// TIA Portal V15.1 export
// export: Created 2024-06-21T08:40:53.4575438Z, ExportSetting WithDefaults, DisplayName Totally Integrated Automation Portal, DisplayVersion V15.1 Update 5, DisplayName TIA Portal Openness, DisplayVersion V15.1 Update 5, DisplayName SINAMICS Startdrive Advanced, DisplayVersion V15.1, DisplayName G130, G150, S120, S150, SINAMICS MV, S210, DisplayVersion V15.1, DisplayName G110M, G120, G120C, G120D, G120P, DisplayVersion V15.1, DisplayName STEP 7 Professional, DisplayVersion V15.1 Update 5, DisplayName STEP 7 Safety, DisplayVersion V15.1, DisplayName WinCC Professional, DisplayVersion V15.1 Update 5, DisplayName SIMATIC Visualization Architect, DisplayVersion V15.1
FUNCTION_BLOCK "LConditionDelay"   // FB1101, FBD
TITLE = LConditionDelay
{ S7_Optimized_Access := 'FALSE' }
VERSION : 0.1
// stored: AutoNumber false, IsIECCheckEnabled false, SetENOAutomatically False, UDAEnableTagReadback false
   VAR_INPUT
      I_Condition { ExternalAccessible := 'False'; ExternalVisible := 'False'; ExternalWritable := 'False'} : Bool;   // Condition
      I_ExtDelayTime { ExternalAccessible := 'False'; ExternalVisible := 'False'; ExternalWritable := 'False'} : DInt;   // External delay time
      I_ActivedExtDelayTime { ExternalAccessible := 'False'; ExternalVisible := 'False'; ExternalWritable := 'False'} : Bool;   // Activated external delay time
      I_HoldCond { ExternalAccessible := 'False'; ExternalVisible := 'False'; ExternalWritable := 'False'} : Bool;   // Hold condition normal open
      I_ResetCond { ExternalAccessible := 'False'; ExternalVisible := 'False'; ExternalWritable := 'False'} : Bool;   // Reset condition normal open
      I_BypassCond { ExternalAccessible := 'False'; ExternalVisible := 'False'; ExternalWritable := 'False'} : Bool;   // Bypass condition normal open
   END_VAR
   VAR_OUTPUT
      O_ConditionDelayed { ExternalAccessible := 'False'; ExternalVisible := 'False'; ExternalWritable := 'False'} : Bool;   // Condition delayed
   END_VAR
   VAR_IN_OUT
      H_HMI : "H_HMI";   // Animation
      H_ConditionDelay : "H_ConditionDelay";   // Animation
   END_VAR
   VAR DB_SPECIFIC
      TimerResult { ExternalAccessible := 'False'; ExternalVisible := 'False'; ExternalWritable := 'False'} : Bool;   // Timer result
      TimerValue { ExternalAccessible := 'False'; ExternalVisible := 'False'; ExternalWritable := 'False'} : DInt;   // Timer value
      TimerValueElapsed { ExternalAccessible := 'False'; ExternalVisible := 'False'; ExternalWritable := 'False'} : DInt;   // Timer value elapsed
      TimerExtValue { ExternalAccessible := 'False'; ExternalVisible := 'False'; ExternalWritable := 'False'} : DInt;   // Timer external value
      PrevExtDelayTime { ExternalAccessible := 'False'; ExternalVisible := 'False'; ExternalWritable := 'False'} : DInt;   // Previous external delay time
   END_VAR
   VAR
      DelayTimer { ExternalAccessible := 'False'; ExternalVisible := 'False'; ExternalWritable := 'False'} : "LTimer";   // Timer
   END_VAR
   VAR DB_SPECIFIC
      Edge { ExternalAccessible := 'False'; ExternalVisible := 'False'; ExternalWritable := 'False'} : Array[1..10] of Bool;   // Edge
   END_VAR
   VAR_TEMP   // added for the SCL form of the ladder/FBD networks
      _w1 : Bool;
      _w2 : Bool;
   END_VAR
BEGIN

REGION Network 1: **** 5.2 - Equations **** Timer External Value
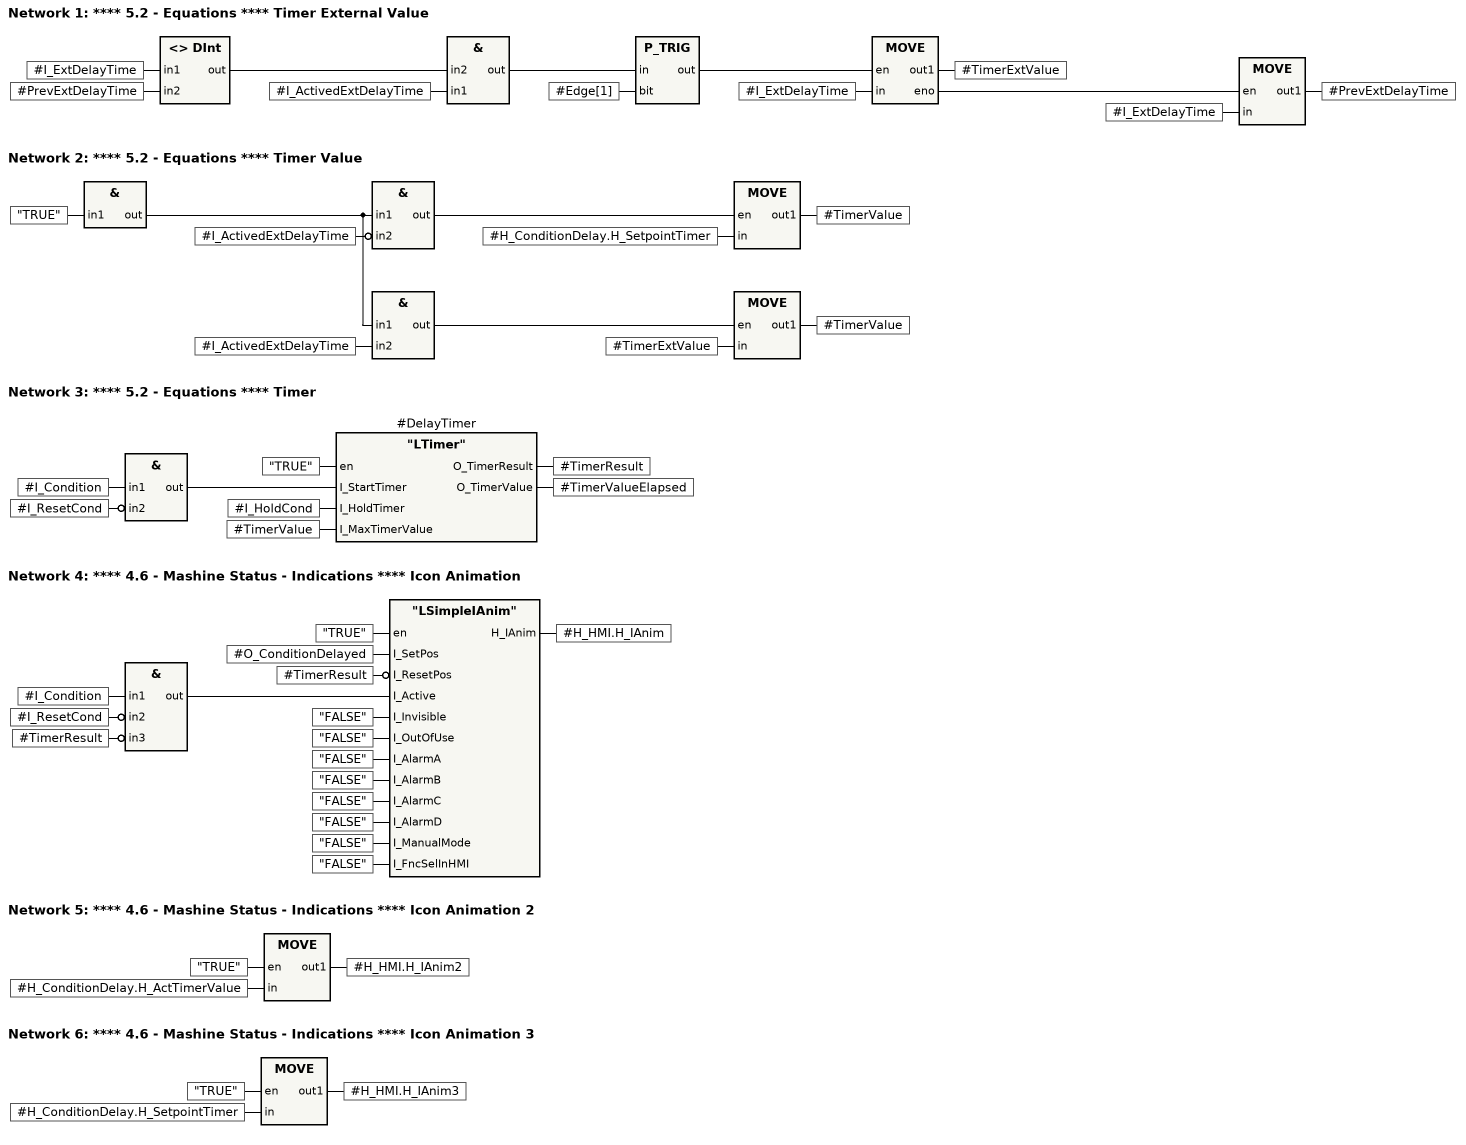
   #_w1 := (#I_ExtDelayTime <> #PrevExtDelayTime) AND #I_ActivedExtDelayTime;
   #_w2 := #_w1 AND NOT #Edge[1];   // rising edge
   #Edge[1] := #_w1;
   IF #_w2 THEN
       #TimerExtValue := #I_ExtDelayTime;
       #PrevExtDelayTime := #I_ExtDelayTime;
   END_IF;
END_REGION

REGION Network 2: **** 5.2 - Equations **** Timer Value
   IF "TRUE" AND NOT #I_ActivedExtDelayTime THEN #TimerValue := #H_ConditionDelay.H_SetpointTimer; END_IF;
   IF "TRUE" AND #I_ActivedExtDelayTime THEN #TimerValue := #TimerExtValue; END_IF;
END_REGION

REGION Network 3: **** 5.2 - Equations **** Timer
   IF "TRUE" THEN
       #DelayTimer(I_StartTimer := #I_Condition AND NOT #I_ResetCond,   // "LTimer"
                   I_HoldTimer := #I_HoldCond,
                   I_MaxTimerValue := #TimerValue,
                   O_TimerResult => #TimerResult,
                   O_TimerValue => #TimerValueElapsed);
   END_IF;
END_REGION

REGION Network 4: **** 4.6 - Mashine Status - Indications **** Icon Animation
   // Icon Animation
   IF "TRUE" THEN
       "LSimpleIAnim"(I_SetPos := #O_ConditionDelayed,
                      I_ResetPos := NOT #TimerResult,
                      I_Active := #I_Condition AND NOT #I_ResetCond AND NOT #TimerResult,
                      I_Invisible := "FALSE",
                      I_OutOfUse := "FALSE",
                      I_AlarmA := "FALSE",
                      I_AlarmB := "FALSE",
                      I_AlarmC := "FALSE",
                      I_AlarmD := "FALSE",
                      I_ManualMode := "FALSE",
                      I_FncSelInHMI := "FALSE",
                      H_IAnim => #H_HMI.H_IAnim);
   END_IF;
END_REGION

REGION Network 5: **** 4.6 - Mashine Status - Indications **** Icon Animation 2
   IF "TRUE" THEN #H_HMI.H_IAnim2 := #H_ConditionDelay.H_ActTimerValue; END_IF;
END_REGION

REGION Network 6: **** 4.6 - Mashine Status - Indications **** Icon Animation 3
   IF "TRUE" THEN #H_HMI.H_IAnim3 := #H_ConditionDelay.H_SetpointTimer; END_IF;
END_REGION

REGION Network 7: **** 4.6 - Machine Status - Indications **** Animation
   // Animation
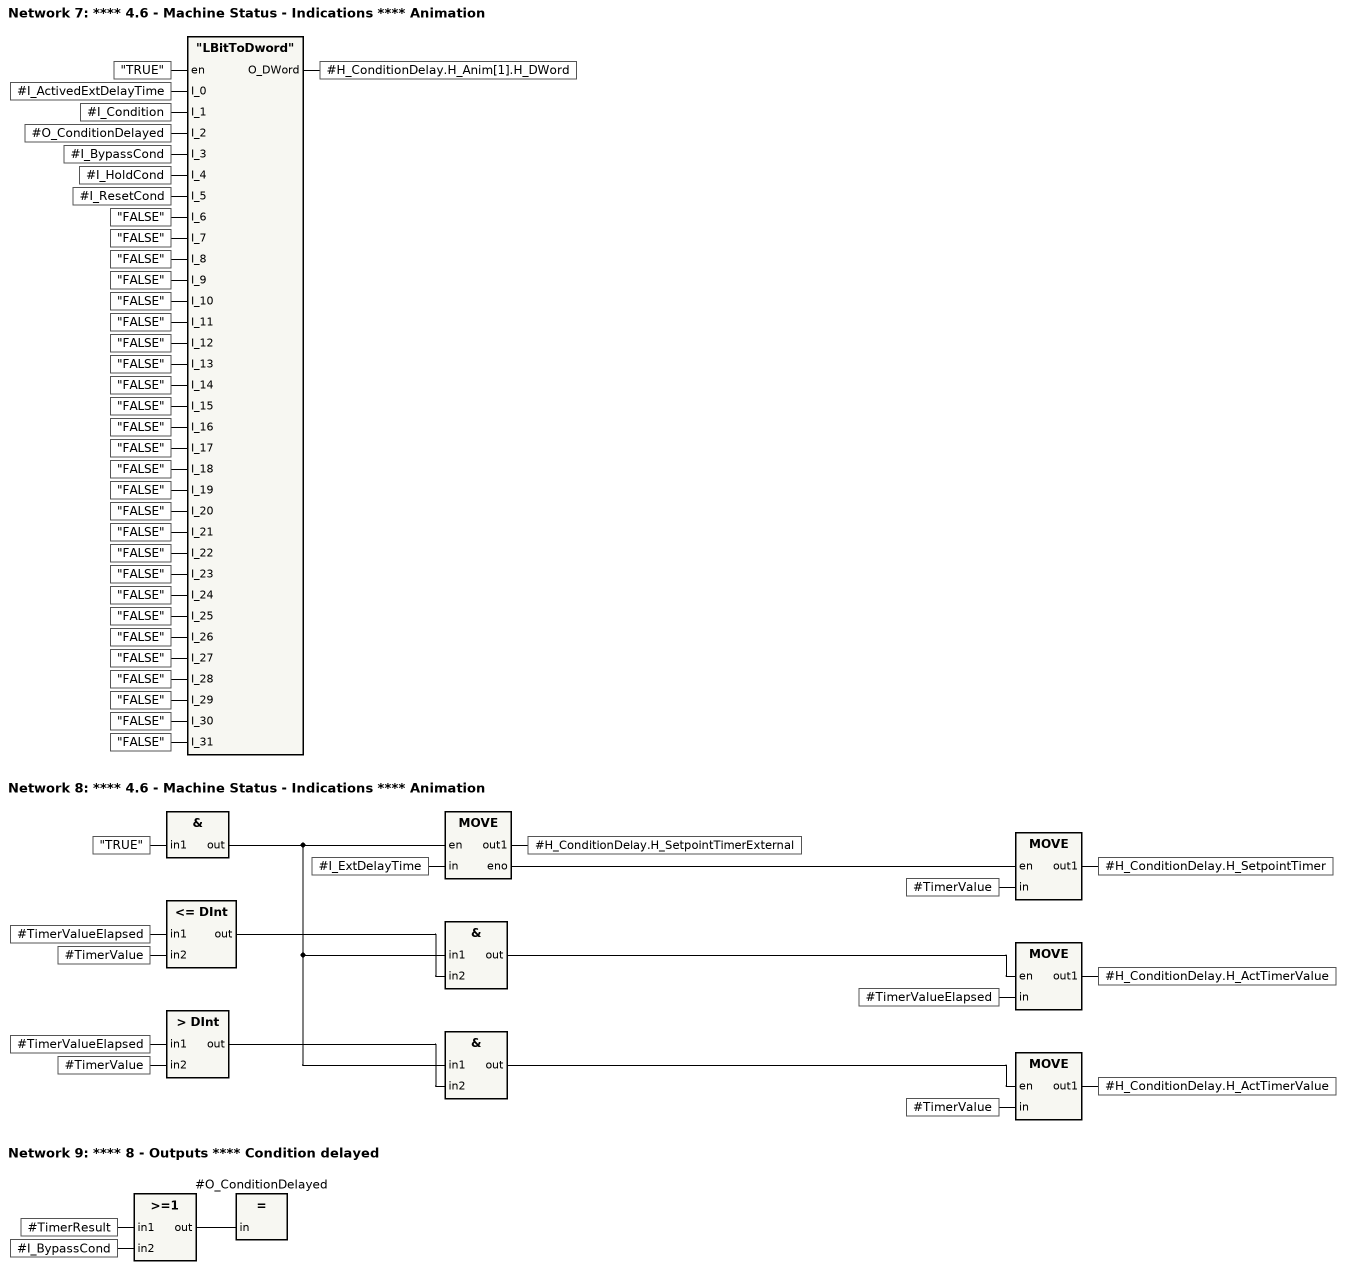
   IF "TRUE" THEN
       "LBitToDword"(I_0 := #I_ActivedExtDelayTime,
                     I_1 := #I_Condition,
                     I_2 := #O_ConditionDelayed,
                     I_3 := #I_BypassCond,
                     I_4 := #I_HoldCond,
                     I_5 := #I_ResetCond,
                     I_6 := "FALSE",
                     I_7 := "FALSE",
                     I_8 := "FALSE",
                     I_9 := "FALSE",
                     I_10 := "FALSE",
                     I_11 := "FALSE",
                     I_12 := "FALSE",
                     I_13 := "FALSE",
                     I_14 := "FALSE",
                     I_15 := "FALSE",
                     I_16 := "FALSE",
                     I_17 := "FALSE",
                     I_18 := "FALSE",
                     I_19 := "FALSE",
                     I_20 := "FALSE",
                     I_21 := "FALSE",
                     I_22 := "FALSE",
                     I_23 := "FALSE",
                     I_24 := "FALSE",
                     I_25 := "FALSE",
                     I_26 := "FALSE",
                     I_27 := "FALSE",
                     I_28 := "FALSE",
                     I_29 := "FALSE",
                     I_30 := "FALSE",
                     I_31 := "FALSE",
                     O_DWord => #H_ConditionDelay.H_Anim[1].H_DWord);
   END_IF;
END_REGION

REGION Network 8: **** 4.6 - Machine Status - Indications **** Animation
   IF "TRUE" THEN
       #H_ConditionDelay.H_SetpointTimerExternal := #I_ExtDelayTime;
       #H_ConditionDelay.H_SetpointTimer := #TimerValue;
   END_IF;
   IF "TRUE" AND (#TimerValueElapsed <= #TimerValue) THEN
       #H_ConditionDelay.H_ActTimerValue := #TimerValueElapsed;
   END_IF;
   IF "TRUE" AND (#TimerValueElapsed > #TimerValue) THEN
       #H_ConditionDelay.H_ActTimerValue := #TimerValue;
   END_IF;
END_REGION

REGION Network 9: **** 8 - Outputs **** Condition delayed
   #O_ConditionDelayed := #TimerResult OR #I_BypassCond;
END_REGION
END_FUNCTION_BLOCK
